FUNCTION_BLOCK FB_MatrixGrow_Test EXTENDS FB_TestSuite
VAR_INPUT
END_VAR
VAR_OUTPUT
END_VAR
VAR
END_VAR

WhenEmptyExpectNoError();
WhenGrownExpectDataRetained();
WhenGrownExpectNewDataFilled();

METHOD PRIVATE WhenEmptyExpectNoError
VAR_INPUT
END_VAR
VAR
	M1 : DynamicMatrix;
	M2 : DynamicMatrix;
	Result : BOOL;
END_VAR
TEST('WhenEmptyExpectNoError');

// @TEST-RUN
M1.Init(0,0);
Result := M2.AsGrown(M1,0,0,0,0,0);

// @TEST-ASSERT
AssertTrue(Result,'Main function call was not successful');

TEST_FINISHED();
END_METHOD

METHOD PRIVATE WhenGrownExpectDataRetained
VAR_INPUT
END_VAR
VAR
	M1 : DynamicMatrix;
	M2 : DynamicMatrix;
	M3 : DynamicMatrix;
	Result : BOOL;
END_VAR
TEST('WhenGrownExpectDataRetained');

// @TEST-RUN
M1.InitMagicSquare(3);
Result := M2.AsGrown(M1,0,0,0,0,0);
M3.AsSubMatrix(M2,1,3,1,3);

// @TEST-ASSERT
AssertTrue(Result,'Main function call was not successful');
AssertTrue(M3.IsEqual(M1),'Old data was not retained');

TEST_FINISHED();
END_METHOD

METHOD PRIVATE WhenGrownExpectNewDataFilled
VAR_INPUT
END_VAR
VAR
	M1 : DynamicMatrix;
	M2 : DynamicMatrix;
	Result : BOOL;
END_VAR
TEST('WhenGrownExpectNewDataFilled');

// @TEST-RUN
M1.InitZeros(3,3);
Result := M2.AsGrown(M1,0,0,1,2,3);

// @TEST-ASSERT
AssertTrue(Result,'Main function call was not successful');
AssertTrue(M2.GetRC(0,0) = 1,'Diagonal data was not filled');
AssertTrue(M2.GetRC(0,1) = 2,'Row data was not filled');
AssertTrue(M2.GetRC(1,0) = 3,'Col data was not filled');

TEST_FINISHED();
END_METHOD

END_FUNCTION_BLOCK

(* stored: Version 1.1.0.1, ProductVersion 3.1.4024.9
   POU FB_MatrixGrow_Test: Id {f905e9c3-df8c-00f6-0b5f-8b95421f6974}, SpecialFunc None
   Method WhenEmptyExpectNoError: Id {f33c6266-2abc-016f-3705-eca988b2ff7d}
   Method WhenGrownExpectDataRetained: Id {d0f572ca-c857-008e-0c86-81984e02dd72}
   Method WhenGrownExpectNewDataFilled: Id {2d28a358-6c94-041e-11f8-956330afdb45} *)
